Fanuc KAREL source: kb00013.KL

-- PROVISIONAL review KL for V770-1; original PC SHA256 19aa980aec278db26d032fdce14f9377aa0d5953915631bc704587a681d8abe7
-- Incomplete behavior may be omitted. Consult companion uncertainty JSON. Do not deploy.
PROGRAM KB00013
%NOLOCKGROUP
BEGIN
  -- UNRESOLVED_PC offsets 5-12; opcodes 9D,23
  -- UNRESOLVED_PC offsets 17-24; opcodes 9D,23
  -- UNRESOLVED_PC offsets 29-51; opcodes 27,22,22,22,31
  -- UNRESOLVED_PC offsets 56-60; opcodes 7F
END KB00013
